// SIMATIC S7-200 project (STEP 7-Micro/WIN), CPU 221 REL 01.10

ORGANIZATION_BLOCK MAIN:OB1
TITLE=PROGRAM COMMENTS
BEGIN
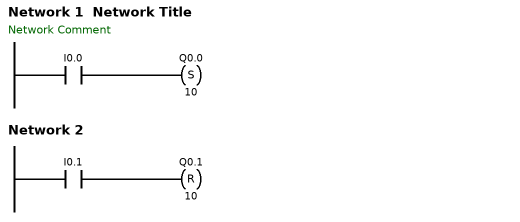
Network 1 // Network Title
// Network Comment
LD     I0.0
S      Q0.0, 10
Network 2
LD     I0.1
R      Q0.1, 10
END_ORGANIZATION_BLOCK
